(* PLC project Unnamed, Unknown Unnamed 1 *)
(* stored: creationDateTime 2026-08-21T10:17:41, modificationDateTime 2026-08-21T10:17:41 *)

PROGRAM main
  VAR
    button AT %IX0.0 : BOOL;
    light AT %QX0.0 : BOOL;
  END_VAR
  VAR
    counter : INT;
  END_VAR

            if button = true then
    light := true;
    counter := true;
else
    light := false;
end_if;
          
END_PROGRAM

CONFIGURATION Config0
  RESOURCE Res0 ON PLC
    TASK task0(INTERVAL := T#20ms, PRIORITY := 1);
    PROGRAM instance0 WITH task0 : main;
  END_RESOURCE
END_CONFIGURATION
